Yaskawa INFORM job: R1-HOME.JBI

/JOB
//NAME R1-HOME
///FOLDERNAME IMPORTANT_JOBS
//POS
///NPOS 1,1,0,0,0,0
///TOOL 0
///POSTYPE ROBOT
///RECTAN
///RCONF 0,0,1,0,0,0,0,0,0,0,0,0,0,0,0,0,0,0,0,0,0,0,0,0
C00000=1690.211,0.059,151.285,-0.1343,-76.2677,0.1330
///RCONF 0,0,0,0,0,0,0,0,0,0,0,0,0,0,0,0,0,0,0,0,0,0,0,0
BC00000=0.397
//INST
///DATE 2024/04/27 12:06
///ATTR SC,RW,RJ
////FRAME ROBOT
///GROUP1 RB1,BS1
NOP
MOVJ C00000 BC00000 VJ=25.00
END
